KUKA KRL program: SET_CP_MAXDELTA.src

&ACCESS RV
&REL 3
&PARAM TEMPLATE = C:\KRC\Roboter\Template\FunctionVorgabe
&PARAM EDITMASK = *
DEFFCT BOOL SET_CP_MAXDELTA( X_VAL:IN, Y_VAL:IN, Z_VAL:IN, A_VAL:IN, B_VAL:IN, C_VAL:IN)

REAL X_VAL, Y_VAL, Z_VAL
REAL A_VAL, B_VAL, C_VAL

$STIFFNESS.CPMAXDELTA.X = X_VAL
$STIFFNESS.CPMAXDELTA.Y = Y_VAL
$STIFFNESS.CPMAXDELTA.Z = Z_VAL
$STIFFNESS.CPMAXDELTA.A = A_VAL
$STIFFNESS.CPMAXDELTA.B = B_VAL
$STIFFNESS.CPMAXDELTA.C = C_VAL

$STIFFNESS.COMMIT = TRUE

RETURN TRUE

ENDFCT
